PROGRAM Mc_01_Units_05
VAR
	HMI_Motion: FB_HMI_Control_NoGroupRef;
	Motion: FB_Motion2way;

	tMessageOffset: UINT;
	tNumMessagesPerRow: UINT;
	
	
	MyAdvanceInterlock: BOOL;
	MyReturnInterlock: BOOL;
	
	MyAutoAdvanceCondition: BOOL;
	MyAutoReturnCondition: BOOL;
	
	myAdvancePrompt: BOOL;
	myReturnPrompt: BOOL;
END_VAR

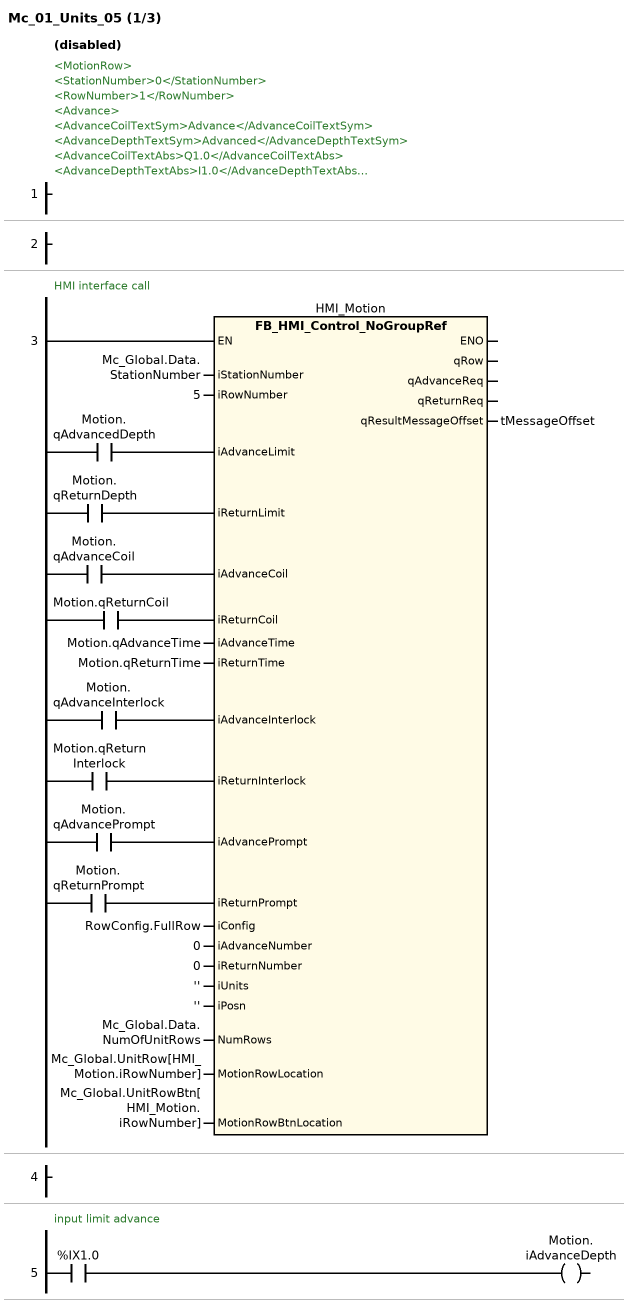
// NETWORK 1 (disabled)
// <MotionRow>
// <StationNumber>0</StationNumber>
// <RowNumber>1</RowNumber>
//   <Advance>
//     <AdvanceCoilTextSym>Advance</AdvanceCoilTextSym>
//     <AdvanceDepthTextSym>Advanced</AdvanceDepthTextSym>
//     <AdvanceCoilTextAbs>Q1.0</AdvanceCoilTextAbs>
//     <AdvanceDepthTextAbs>I1.0</AdvanceDepthTextAbs>
//     <ManSeq>1</ManSeq>
//   </Advance>
//   <Return>
//     <ReturnCoilTextSym>Return</ReturnCoilTextSym>
//     <ReturnDepthTextSym>Returned</ReturnDepthTextSym>
//     <ReturnCoilTextAbs>Q1.1</ReturnCoilTextAbs>
//     <ReturnDepthTextAbs>I1.1</ReturnDepthTextAbs>
//    <ManSeq>2</ManSeq>
//   </Return>
//   <Motion>
//     <NameSym>Station Lighting</NameSym>
//     <NameAbs>KF1</NameAbs>
//   </Motion>
// </MotionRow>

// NETWORK 2

// NETWORK 3
// HMI interface call
HMI_Motion(
    iStationNumber := Mc_Global.Data.StationNumber,
    iRowNumber := 5,
    iAdvanceLimit := Motion.qAdvancedDepth,
    iReturnLimit := Motion.qReturnDepth,
    iAdvanceCoil := Motion.qAdvanceCoil,
    iReturnCoil := Motion.qReturnCoil,
    iAdvanceTime := Motion.qAdvanceTime,
    iReturnTime := Motion.qReturnTime,
    iAdvanceInterlock := Motion.qAdvanceInterlock,
    iReturnInterlock := Motion.qReturnInterlock,
    iAdvancePrompt := Motion.qAdvancePrompt,
    iReturnPrompt := Motion.qReturnPrompt,
    iConfig := RowConfig.FullRow,
    iAdvanceNumber := 0,
    iReturnNumber := 0,
    iUnits := '',
    iPosn := '',
    NumRows := Mc_Global.Data.NumOfUnitRows,
    MotionRowLocation := Mc_Global.UnitRow[HMI_Motion.iRowNumber],
    MotionRowBtnLocation := Mc_Global.UnitRowBtn[HMI_Motion.iRowNumber],
    qResultMessageOffset => tMessageOffset); // FB_HMI_Control_NoGroupRef

// NETWORK 4

// NETWORK 5
// input limit advance
Motion.iAdvanceDepth := %IX1.0;

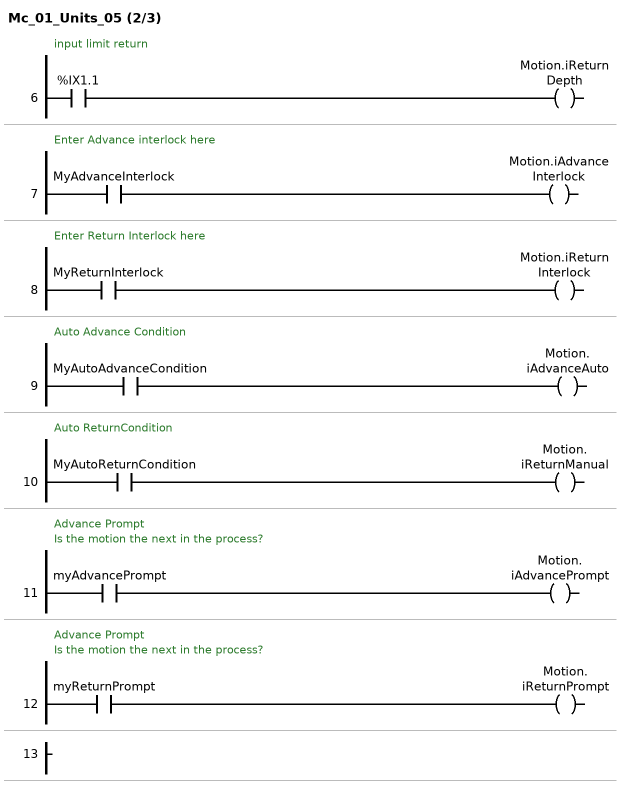
// NETWORK 6
// input limit return
Motion.iReturnDepth := %IX1.1;

// NETWORK 7
// Enter Advance interlock here
Motion.iAdvanceInterlock := MyAdvanceInterlock;

// NETWORK 8
// Enter Return Interlock here
Motion.iReturnInterlock := MyReturnInterlock;

// NETWORK 9
// Auto Advance Condition
Motion.iAdvanceAuto := MyAutoAdvanceCondition;

// NETWORK 10
// Auto ReturnCondition
Motion.iReturnManual := MyAutoReturnCondition;

// NETWORK 11
// Advance Prompt
// Is the motion the next in the process?
Motion.iAdvancePrompt := myAdvancePrompt;

// NETWORK 12
// Advance Prompt
// Is the motion the next in the process?
Motion.iReturnPrompt := myReturnPrompt;

// NETWORK 13

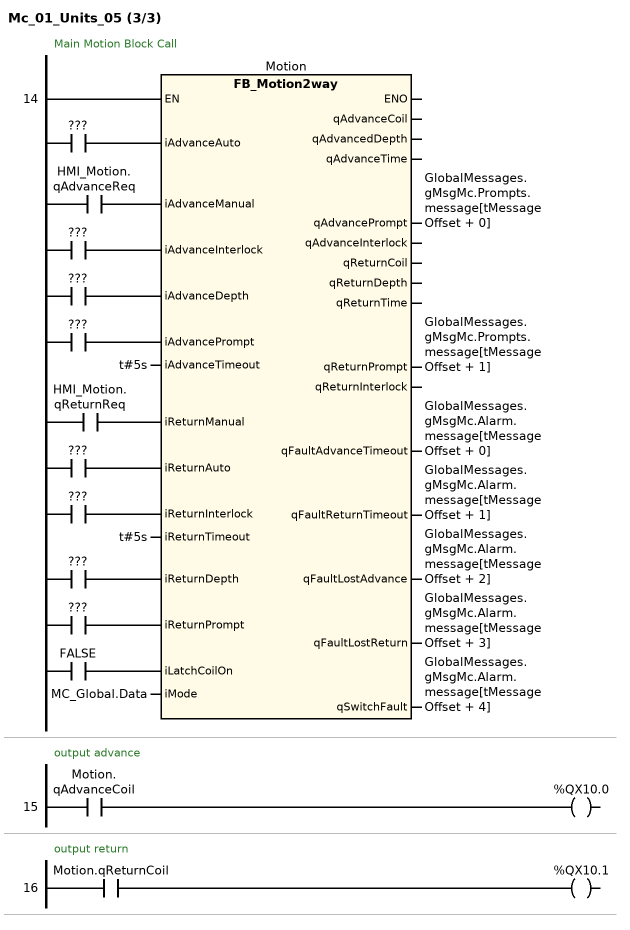
// NETWORK 14
// Main Motion Block Call
Motion(
    iAdvanceManual := HMI_Motion.qAdvanceReq,
    iAdvanceTimeout := t#5s,
    iReturnManual := HMI_Motion.qReturnReq,
    iReturnTimeout := t#5s,
    iLatchCoilOn := FALSE,
    iMode := MC_Global.Data,
    qAdvancePrompt => GlobalMessages.gMsgMc.Prompts.message[tMessageOffset + 0],
    qReturnPrompt => GlobalMessages.gMsgMc.Prompts.message[tMessageOffset + 1],
    qFaultAdvanceTimeout => GlobalMessages.gMsgMc.Alarm.message[tMessageOffset + 0],
    qFaultReturnTimeout => GlobalMessages.gMsgMc.Alarm.message[tMessageOffset + 1],
    qFaultLostAdvance => GlobalMessages.gMsgMc.Alarm.message[tMessageOffset + 2],
    qFaultLostReturn => GlobalMessages.gMsgMc.Alarm.message[tMessageOffset + 3],
    qSwitchFault => GlobalMessages.gMsgMc.Alarm.message[tMessageOffset + 4]); // FB_Motion2way

// NETWORK 15
// output advance
%QX10.0 := Motion.qAdvanceCoil;

// NETWORK 16
// output return
%QX10.1 := Motion.qReturnCoil;

END_PROGRAM

(* stored: Version 1.1.0.1, ProductVersion 3.1.4024.12
   POU Mc_01_Units_05: Id {24a87102-c53b-41c9-802a-4e15622f2e6d}, SpecialFunc None *)
